FUNCTION_BLOCK DeserializerGarbageCollector_TestSuite EXTENDS TcUnit.FB_TestSuite

TestRegister();
TestExecute();
TestDeregister();

METHOD PUBLIC TestDeregister
VAR
	deserializerGarbageCollector : DeserializerGarbageCollector;
	mockDisposableDeserializer : MockDisposableDeserializer;
END_VAR
TEST('TestDeregister');

deserializerGarbageCollector.Register(mockDisposableDeserializer);
deserializerGarbageCollector.Deregister(mockDisposableDeserializer);
deserializerGarbageCollector.Execute();

AssertFalse(
	Condition := mockDisposableDeserializer.IsDisposed,
	Message := 'Did not deregister the deserializer, which resulted in it disposing.'
);

TEST_FINISHED();
END_METHOD

METHOD PUBLIC TestExecute
VAR
	deserializerGarbageCollector : DeserializerGarbageCollector;
	mockDisposableDeserializer : MockDisposableDeserializer;
END_VAR
TEST('TestExecute');

deserializerGarbageCollector.Register(mockDisposableDeserializer);
deserializerGarbageCollector.Execute();

AssertTrue(
	Condition := mockDisposableDeserializer.IsDisposed,
	Message := 'Did not dispose of the registered Deserializer'
);

TEST_FINISHED();
END_METHOD

METHOD PUBLIC TestRegister
VAR
	deserializerGarbageCollector : DeserializerGarbageCollector;
	mockDisposableDeserializer : MockDisposableDeserializer;
END_VAR
TEST('TestRegister');

deserializerGarbageCollector.Register(mockDisposableDeserializer);
deserializerGarbageCollector.Execute();

AssertTrue(
	Condition := mockDisposableDeserializer.IsDisposed,
	Message := 'Did not register the deserializer'
);

TEST_FINISHED();
END_METHOD

END_FUNCTION_BLOCK

(* stored: Version 1.1.0.1, ProductVersion 3.1.4024.12
   POU DeserializerGarbageCollector_TestSuite: Id {5c1b502e-8c5a-0977-1832-83cbd83f5a96}, SpecialFunc None
   Method TestDeregister: Id {4c7abe54-ebbd-0614-0e32-1c9671dc368d}
   Method TestExecute: Id {28f2f5a5-c536-0c12-36a3-cbae763d201e}
   Method TestRegister: Id {0446081a-c175-097d-227d-525d61b652b7} *)
